FUNCTION_BLOCK DEMO_Operator (* Automatic operator for demos: occupy, reset in Production, start, wait for Complete, new vial, pause, repeat while Enable; clears the unit after an abort *)
  (* Standard: 61499-2 *)
  (* Version 2.0, 2026-09-27, Project contributors, Filling cell reference model *)
  PACKAGE fillingcell;
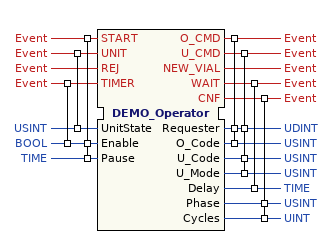
  EVENT_INPUT
    START WITH Enable, Pause;
    UNIT WITH UnitState;
    REJ;
    TIMER WITH Enable;
  END_EVENT
  EVENT_OUTPUT
    O_CMD WITH Requester, O_Code;
    U_CMD WITH Requester, U_Code, U_Mode;
    NEW_VIAL;
    WAIT WITH Delay;
    CNF WITH Phase, Cycles;
  END_EVENT
  VAR_INPUT
    UnitState : USINT;
    Enable : BOOL := TRUE;
    Pause : TIME := T#2s;
  END_VAR
  VAR_OUTPUT
    Requester : UDINT := 1;
    O_Code : USINT;
    U_Code : USINT;
    U_Mode : USINT;
    Delay : TIME;
    Phase : USINT;
    Cycles : UINT;
  END_VAR
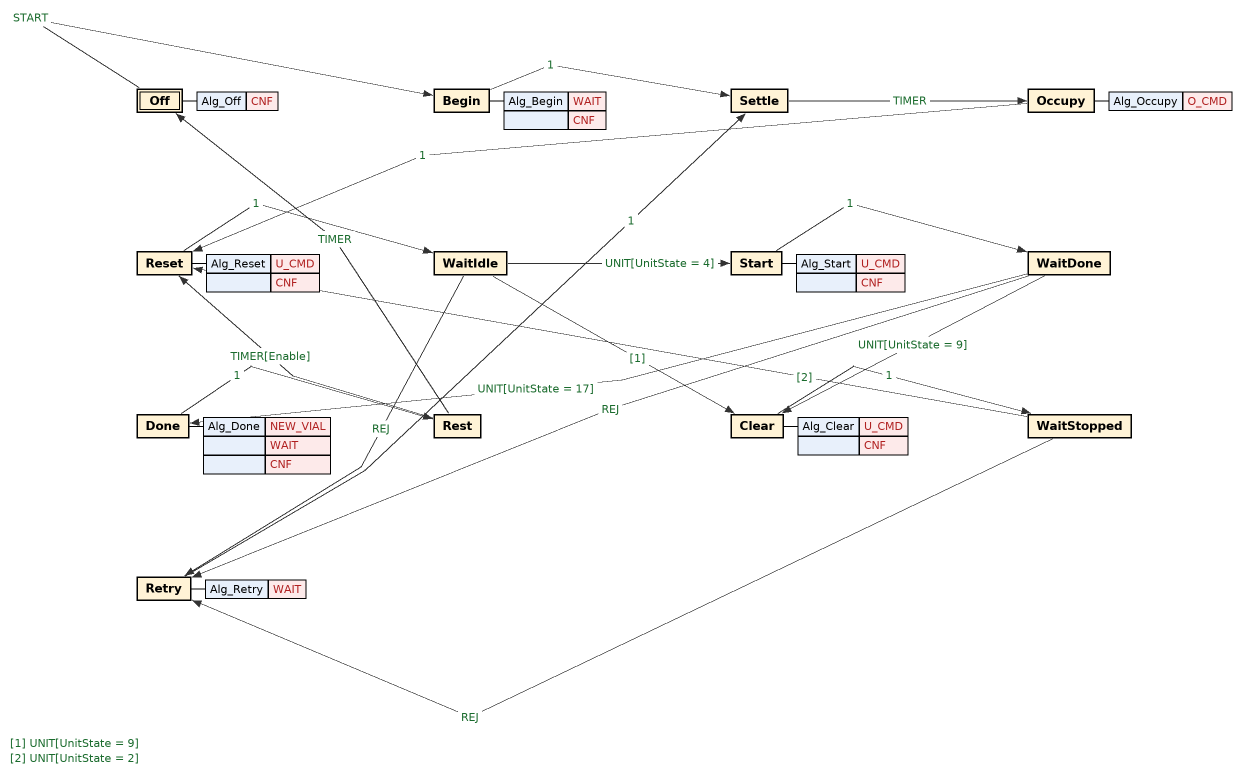
  EC_STATES
    Off : Alg_Off -> CNF;
    Begin : Alg_Begin -> WAIT, -> CNF;
    Settle;
    Occupy : Alg_Occupy -> O_CMD;
    Reset : Alg_Reset -> U_CMD, -> CNF;
    WaitIdle;
    Start : Alg_Start -> U_CMD, -> CNF;
    WaitDone;
    Done : Alg_Done -> NEW_VIAL, -> WAIT, -> CNF;
    Rest;
    Clear : Alg_Clear -> U_CMD, -> CNF;
    WaitStopped;
    Retry : Alg_Retry -> WAIT;
  END_STATES
  EC_TRANSITIONS
    Off TO Begin := START;
    Begin TO Settle := 1;
    Settle TO Occupy := TIMER;
    Occupy TO Reset := 1;
    Reset TO WaitIdle := 1;
    WaitIdle TO Start := UNIT[UnitState = 4];
    WaitIdle TO Clear := UNIT[UnitState = 9];
    WaitIdle TO Retry := REJ;
    Start TO WaitDone := 1;
    WaitDone TO Done := UNIT[UnitState = 17];
    WaitDone TO Clear := UNIT[UnitState = 9];
    WaitDone TO Retry := REJ;
    Done TO Rest := 1;
    Rest TO Reset := TIMER[Enable];
    Rest TO Off := TIMER;
    Clear TO WaitStopped := 1;
    WaitStopped TO Reset := UNIT[UnitState = 2];
    WaitStopped TO Retry := REJ;
    Retry TO Settle := 1;
  END_TRANSITIONS
  ALGORITHM Alg_Off IN ST:
Phase := 0;
  END_ALGORITHM
  ALGORITHM Alg_Begin IN ST:
Phase := 1;
Delay := T#1s;
  END_ALGORITHM
  ALGORITHM Alg_Occupy IN ST:
O_Code := 1;
  END_ALGORITHM
  ALGORITHM Alg_Reset IN ST:
U_Code := 1;
U_Mode := 0;
Phase := 2;
  END_ALGORITHM
  ALGORITHM Alg_Start IN ST:
U_Code := 2;
Phase := 3;
  END_ALGORITHM
  ALGORITHM Alg_Done IN ST:
Cycles := Cycles + 1;
Delay := Pause;
Phase := 4;
  END_ALGORITHM
  ALGORITHM Alg_Clear IN ST:
U_Code := 7;
Phase := 5;
  END_ALGORITHM
  ALGORITHM Alg_Retry IN ST:
Delay := T#1s;
  END_ALGORITHM
END_FUNCTION_BLOCK
